LIN {X 0,Y 88.152,Z 588.258,A -85,B 0,C 180,E1 -30791.719,E2 -30791.719} C_VEL
LIN {X 0,Y 88.811,Z 591.453,A -85,B 0,C 180,E1 -30797.684,E2 -30797.684} C_VEL
LIN {X 0,Y 89.501,Z 594.103,A -85,B 0,C 180,E1 -30801.091,E2 -30801.091} C_VEL
LIN {X 0,Y 87.194,Z 611.74,A -85,B 0,C 180,E1 -30802.089,E2 -30802.089} C_VEL
LIN {X 0,Y 84.33,Z 623.957,A -85,B 0,C 180,E1 -30803.084,E2 -30803.084} C_VEL
LIN {X 0,Y 82.485,Z 629.573,A -85,B 0,C 180,E1 -30803.214,E2 -30803.214} C_VEL
LIN {X 0,Y 78.532,Z 638.576,A -85,B 0,C 180,E1 -30802.242,E2 -30802.242} C_VEL
LIN {X 0,Y 73.895,Z 647.262,A -85,B 0,C 180,E1 -30801.238,E2 -30801.238} C_VEL
LIN {X 0,Y 70.936,Z 652.382,A -85,B 0,C 180,E1 -30801.459,E2 -30801.459} C_VEL
LIN {X 0,Y 63.345,Z 664.109,A -85,B 0,C 180,E1 -30803.776,E2 -30803.776} C_VEL
LIN {X 0,Y 55.091,Z 674.339,A -85,B 0,C 180,E1 -30806.777,E2 -30806.777} C_VEL
LIN {X 0,Y 46.982,Z 682.675,A -85,B 0,C 180,E1 -30810.697,E2 -30810.697} C_VEL
LIN {X 0,Y 37.512,Z 690.88,A -85,B 0,C 180,E1 -30817.256,E2 -30817.256} C_VEL
LIN {X 0,Y 28.021,Z 697.992,A -85,B 0,C 180,E1 -30828.795,E2 -30828.795} C_VEL
LIN {X 0,Y 20.283,Z 703.592,A -85,B 0,C 180,E1 -30849.762,E2 -30849.762} C_VEL
LIN {X 0,Y 17.277,Z 707.59,A -85,B 0,C 180,E1 -30881.775,E2 -30881.775} C_VEL
LIN {X 0,Y 17.637,Z 708.712,A -85,B 0,C 180,E1 -30893.524,E2 -30893.524} C_VEL
LIN {X 0,Y 18.657,Z 710.303,A -85,B 0,C 180,E1 -30911.128,E2 -30911.128} C_VEL
LIN {X 0,Y 19.957,Z 714.833,A -85,B 0,C 180,E1 -30980.627,E2 -30980.627} C_VEL
LIN {X 0,Y 26.819,Z 716.625,A -85,B 0,C 180,E1 -30998.133,E2 -30998.133} C_VEL
LIN {X 0,Y 28.963,Z 717.13,A -85,B 0,C 180,E1 -31003.25,E2 -31003.25} C_VEL
LIN {X 0,Y 24.466,Z 716.245,A -85,B 0,C 180,E1 -31014.901,E2 -31014.901} C_VEL
LIN {X 0,Y 18.055,Z 713.675,A -85,B 0,C 180,E1 -31038.739,E2 -31038.739} C_VEL
LIN {X 0,Y 16.766,Z 710.04,A -85,B 0,C 180,E1 -31074.739,E2 -31074.739} C_VEL
LIN {X 0,Y 21.785,Z 705.308,A -85,B 0,C 180,E1 -31103.703,E2 -31103.703} C_VEL
LIN {X 0,Y 31.605,Z 698.175,A -85,B 0,C 180,E1 -31120.856,E2 -31120.856} C_VEL
LIN {X 0,Y 41.263,Z 690.484,A -85,B 0,C 180,E1 -31128.25,E2 -31128.25} C_VEL
LIN {X 0,Y 49.666,Z 682.67,A -85,B 0,C 180,E1 -31132.01,E2 -31132.01} C_VEL
LIN {X 0,Y 58.237,Z 673.208,A -85,B 0,C 180,E1 -31134.493,E2 -31134.493} C_VEL
LIN {X 0,Y 66.021,Z 662.65,A -85,B 0,C 180,E1 -31136.197,E2 -31136.197} C_VEL
LIN {X 0,Y 72.978,Z 650.921,A -85,B 0,C 180,E1 -31137.395,E2 -31137.395} C_VEL
LIN {X 0,Y 78.7,Z 638.303,A -85,B 0,C 180,E1 -31138.299,E2 -31138.299} C_VEL
LIN {X 0,Y 82.973,Z 625.381,A -85,B 0,C 180,E1 -31138.962,E2 -31138.962} C_VEL
LIN {X 0,Y 84.901,Z 616.76,A -85,B 0,C 180,E1 -31139.792,E2 -31139.792} C_VEL
LIN {X 0,Y 87.219,Z 598.951,A -85,B 0,C 180,E1 -31141.587,E2 -31141.587} C_VEL
LIN {X 0,Y 87.462,Z 596.724,A -85,B 0,C 180,E1 -31141.798,E2 -31141.798} C_VEL
LIN {X 0,Y 87.293,Z 595.1,A -85,B 0,C 180,E1 -31144.616,E2 -31144.616} C_VEL
LIN {X 0,Y 87.21,Z 595.13,A -85,B 0,C 180,E1 -31150.69,E2 -31150.69} C_VEL
LIN {X 0,Y 87.678,Z 598.333,A -85,B 0,C 180,E1 -31156.6,E2 -31156.6} C_VEL
LIN {X 0,Y 87.666,Z 598.92,A -85,B 0,C 180,E1 -31156.868,E2 -31156.868} C_VEL
LIN {X 0,Y 85.384,Z 614.288,A -85,B 0,C 180,E1 -31157.609,E2 -31157.609} C_VEL
LIN {X 0,Y 82.053,Z 627.05,A -85,B 0,C 180,E1 -31158.562,E2 -31158.562} C_VEL
LIN {X 0,Y 77.476,Z 639.359,A -85,B 0,C 180,E1 -31159.784,E2 -31159.784} C_VEL
LIN {X 0,Y 71.637,Z 651.188,A -85,B 0,C 180,E1 -31161.278,E2 -31161.278} C_VEL
LIN {X 0,Y 70.936,Z 652.382,A -85,B 0,C 180,E1 -31161.459,E2 -31161.459} C_VEL
LIN {X 0,Y 67.772,Z 657.428,A -85,B 0,C 180,E1 -31161.743,E2 -31161.743} C_VEL
LIN {X 0,Y 61.881,Z 665.341,A -85,B 0,C 180,E1 -31160.761,E2 -31160.761} C_VEL
LIN {X 0,Y 55.47,Z 672.809,A -85,B 0,C 180,E1 -31159.674,E2 -31159.674} C_VEL
LIN {X 0,Y 51.457,Z 677.08,A -85,B 0,C 180,E1 -31160.1,E2 -31160.1} C_VEL
LIN {X 0,Y 42.104,Z 685.894,A -85,B 0,C 180,E1 -31163.397,E2 -31163.397} C_VEL
LIN {X 0,Y 32.034,Z 693.65,A -85,B 0,C 180,E1 -31168.696,E2 -31168.696} C_VEL
LIN {X 0,Y 22.598,Z 699.755,A -85,B 0,C 180,E1 -31177.735,E2 -31177.735} C_VEL
LIN {X 0,Y 13.761,Z 704.954,A -85,B 0,C 180,E1 -31199.345,E2 -31199.345} C_VEL
LIN {X 0,Y 10.335,Z 708.863,A -85,B 0,C 180,E1 -31249.947,E2 -31249.947} C_VEL
LIN {X 0,Y 10.358,Z 710.18,A -85,B 0,C 180,E1 -31272.817,E2 -31272.817} C_VEL
LIN {X 0,Y 16.386,Z 714.421,A -85,B 0,C 180,E1 -31360.946,E2 -31360.946} C_VEL
LIN {X 0,Y 16.071,Z 714.305,A -85,B 0,C 180,E1 -31368.703,E2 -31368.703} C_VEL
LIN {X 0,Y 9.631,Z 711.284,A -85,B 0,C 180,E1 -31409.93,E2 -31409.93} C_VEL
LIN {X 0,Y 13.468,Z 706.799,A -85,B 0,C 180,E1 -31468.532,E2 -31468.532} C_VEL
LIN {X 0,Y 23.279,Z 700.982,A -85,B 0,C 180,E1 -31488.72,E2 -31488.72} C_VEL
LIN {X 0,Y 33.464,Z 694.177,A -85,B 0,C 180,E1 -31495.728,E2 -31495.728} C_VEL
LIN {X 0,Y 44.041,Z 685.665,A -85,B 0,C 180,E1 -31499.208,E2 -31499.208} C_VEL
LIN {X 0,Y 52.703,Z 677.209,A -85,B 0,C 180,E1 -31500.838,E2 -31500.838} C_VEL
LIN {X 0,Y 61.519,Z 666.626,A -85,B 0,C 180,E1 -31501.974,E2 -31501.974} C_VEL
LIN {X 0,Y 69.469,Z 654.693,A -85,B 0,C 180,E1 -31502.74,E2 -31502.74} C_VEL
LIN {X 0,Y 75.66,Z 642.682,A -85,B 0,C 180,E1 -31503.245,E2 -31503.245} C_VEL
LIN {X 0,Y 80.692,Z 629.612,A -85,B 0,C 180,E1 -31503.746,E2 -31503.746} C_VEL
LIN {X 0,Y 82.829,Z 622.31,A -85,B 0,C 180,E1 -31504.026,E2 -31504.026} C_VEL
LIN {X 0,Y 85.428,Z 608.969,A -85,B 0,C 180,E1 -31505.383,E2 -31505.383} C_VEL
LIN {X 0,Y 86.309,Z 602.163,A -85,B 0,C 180,E1 -31505.99,E2 -31505.99} C_VEL
LIN {X 0,Y 86.29,Z 602.097,A -85,B 0,C 180,E1 -31509.747,E2 -31509.747} C_VEL
LIN {X 0,Y 86.327,Z 603.412,A -85,B 0,C 180,E1 -31512.368,E2 -31512.368} C_VEL
LIN {X 0,Y 84.063,Z 616.68,A -85,B 0,C 180,E1 -31512.971,E2 -31512.971} C_VEL
LIN {X 0,Y 80.344,Z 629.869,A -85,B 0,C 180,E1 -31513.814,E2 -31513.814} C_VEL
LIN {X 0,Y 75.389,Z 642.267,A -85,B 0,C 180,E1 -31514.754,E2 -31514.754} C_VEL
LIN {X 0,Y 69.394,Z 653.585,A -85,B 0,C 180,E1 -31515.856,E2 -31515.856} C_VEL
LIN {X 0,Y 61.703,Z 665.082,A -85,B 0,C 180,E1 -31517.499,E2 -31517.499} C_VEL
LIN {X 0,Y 54.003,Z 674.399,A -85,B 0,C 180,E1 -31519.387,E2 -31519.387} C_VEL
LIN {X 0,Y 51.457,Z 677.08,A -85,B 0,C 180,E1 -31520.1,E2 -31520.1} C_VEL
LIN {X 0,Y 47.261,Z 681.227,A -85,B 0,C 180,E1 -31520.597,E2 -31520.597} C_VEL
LIN {X 0,Y 39.781,Z 687.659,A -85,B 0,C 180,E1 -31519.082,E2 -31519.082} C_VEL
LIN {X 0,Y 31.863,Z 693.504,A -85,B 0,C 180,E1 -31516.798,E2 -31516.798} C_VEL
LIN {X 0,Y 26.898,Z 696.732,A -85,B 0,C 180,E1 -31517.029,E2 -31517.029} C_VEL
LIN {X 0,Y 15.275,Z 703.15,A -85,B 0,C 180,E1 -31523.157,E2 -31523.157} C_VEL
LIN {X 0,Y 5.297,Z 707.703,A -85,B 0,C 180,E1 -31548.614,E2 -31548.614} C_VEL
LIN {X 0,Y 3.25,Z 709.003,A -85,B 0,C 180,E1 -31590.207,E2 -31590.207} C_VEL
LIN {X 0,Y 2.06,Z 710.164,A -85,B 0,C 180,E1 -31680.072,E2 -31680.072} C_VEL
LIN {X 0,Y 2.694,Z 710.477,A -85,B 0,C 180,E1 -31706.272,E2 -31706.272} C_VEL
LIN {X 0,Y 2.383,Z 710.002,A -85,B 0,C 180,E1 -31769.717,E2 -31769.717} C_VEL
LIN {X 0,Y 11.686,Z 705.317,A -85,B 0,C 180,E1 -31861.301,E2 -31861.301} C_VEL
LIN {X 0,Y 22.979,Z 699.474,A -85,B 0,C 180,E1 -31866.544,E2 -31866.544} C_VEL
LIN {X 0,Y 33.699,Z 692.554,A -85,B 0,C 180,E1 -31868.007,E2 -31868.007} C_VEL
LIN {X 0,Y 44.115,Z 684.265,A -85,B 0,C 180,E1 -31868.487,E2 -31868.487} C_VEL
LIN {X 0,Y 53.286,Z 675.263,A -85,B 0,C 180,E1 -31868.521,E2 -31868.521} C_VEL
LIN {X 0,Y 62.18,Z 664.445,A -85,B 0,C 180,E1 -31868.586,E2 -31868.586} C_VEL
LIN {X 0,Y 69.289,Z 653.704,A -85,B 0,C 180,E1 -31868.596,E2 -31868.596} C_VEL
LIN {X 0,Y 75.515,Z 641.687,A -85,B 0,C 180,E1 -31868.628,E2 -31868.628} C_VEL
LIN {X 0,Y 78.194,Z 635.297,A -85,B 0,C 180,E1 -31868.693,E2 -31868.693} C_VEL
LIN {X 0,Y 78.251,Z 635.126,A -85,B 0,C 180,E1 -31868.963,E2 -31868.963} C_VEL
LIN {X 0,Y 73.043,Z 646.744,A -85,B 0,C 180,E1 -31869.577,E2 -31869.577} C_VEL
LIN {X 0,Y 66.945,Z 657.38,A -85,B 0,C 180,E1 -31870.259,E2 -31870.259} C_VEL
LIN {X 0,Y 59.081,Z 668.283,A -85,B 0,C 180,E1 -31871.135,E2 -31871.135} C_VEL
LIN {X 0,Y 50.335,Z 678.072,A -85,B 0,C 180,E1 -31872.276,E2 -31872.276} C_VEL
LIN {X 0,Y 41.574,Z 686.127,A -85,B 0,C 180,E1 -31873.656,E2 -31873.656} C_VEL
LIN {X 0,Y 31.043,Z 694.066,A -85,B 0,C 180,E1 -31875.89,E2 -31875.89} C_VEL
LIN {X 0,Y 26.898,Z 696.732,A -85,B 0,C 180,E1 -31877.029,E2 -31877.029} C_VEL
LIN {X 0,Y 26.898,Z 696.732,A -85,B 0,C 180,E1 -31877.029,E2 -31877.029}

QRS_NEXT_CUT()

QRS_NEXT()
QRS_HOME()

END
